# EPICS substitutions: vacuum/MAIN_TRUNK/db/l411_agilent4uhv.substitutions
# Agilent4UHV substitutions file

file db/agilent4uhv.db
{
     pattern {LOCA,			DEV,			PORT,		ADDR,	TIMEOUT}
     		{HL4,			VL411_1,		4uhv_1,		0,		0.2}
     		{HL4,			VL411_2,		4uhv_2,		0,		0.2}
}

file db/agilent4uhv_alias.db
{
     pattern {LOCA,			DEV,			SUB1,				SUB2,				SUB3,					SUB4,				PORT,		ADDR,	TIMEOUT}
     		 {HL4,			VL411_1,		IP01:L411_Acc601,		IP02:L411_Acc602,		IP03:L411_Acc603,			IP04:L411_Acc604,		4uhv_1,		0,		0.2}
		 {HL4,			VL411_2,		IP05:L411_Acc605,		IP06:L411_Wave601,	IP07:L411_Kly601,			IP08:Empty,			4uhv_2,		0,		0.2}
}
